{attribute 'qualified_only'}
TYPE
    E_PullOutConveyorPosition :
    (
        Undefined := 0,
        I3_Slide, // The left side when facing the machine’s operating side.
        I4_Slide  // The right side when facing the machine’s operating side.
    );
END_TYPE

(* stored: Version 1.1.0.1, ProductVersion 3.1.4024.13
   DUT E_PullOutConveyorPosition: Id {74dcb94a-105e-4d9c-878c-7f302b131778} *)
